FUNCTION_BLOCK CSV_WRITER_7 (* Service Interface Function Block Type *)
  PACKAGE eclipse4diac::utils;
  {SET_ATTRIBUTE(eclipse4diac::core::GenericClassName, 'GEN_CSV_WRITER')}
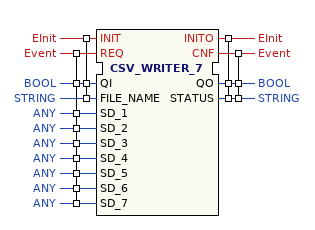
  EVENT_INPUT
    INIT : EInit WITH QI, FILE_NAME; (* Service Initialization *)
    REQ WITH QI, SD_1, SD_2, SD_3, SD_4, SD_5, SD_6, SD_7; (* Service Request *)
  END_EVENT
  EVENT_OUTPUT
    INITO : EInit WITH QO, STATUS; (* Initialization Confirm *)
    CNF WITH QO, STATUS; (* Confirmation of Requested Service *)
  END_EVENT
  VAR_INPUT
    QI : BOOL; (* Event Input Qualifier *)
    FILE_NAME : STRING; (* Service Parameters *)
    SD_1 : ANY; (* Output data to resource *)
    SD_2 : ANY;
    SD_3 : ANY;
    SD_4 : ANY;
    SD_5 : ANY;
    SD_6 : ANY;
    SD_7 : ANY;
  END_VAR
  VAR_OUTPUT
    QO : BOOL; (* Event Output Qualifier *)
    STATUS : STRING; (* File access status *)
  END_VAR
END_FUNCTION_BLOCK
